{attribute addProperty BoxType "EL2212-0000-0018"}
{attribute addProperty Id "StatusAT %I*Status_5D7D7DCC162"}
{attribute addProperty CRC "2034971558"}
{attribute addProperty SizeInBites "16"}
{attribute addProperty SizeInBytes "2"}
TYPE DOX_Status_Channel_794B33A6 :
STRUCT
	{attribute addProperty Name "Status"}
	Status AT %I* : Status_5D7D7DCC;
END_STRUCT
END_TYPE

(* stored: Version 1.2.0.0, ProductVersion 3.1.4024.9
   DUT DOX_Status_Channel_794B33A6: Id {880a3785-d79a-4878-9cda-cea45a8cc4b3} *)
